// TIA Portal V20 export
VAR_GLOBAL   // PLC tag table "EasyBOX"
   I_OUT_TRAY1 AT %I31.0 : Bool;
   I_OUT_TRAY2 AT %I31.1 : Bool;
   I_OUT_TRAY3 AT %I31.2 : Bool;
   I_OUT_TRAY4 AT %I31.3 : Bool;
   I_OUT_TRAY5 AT %I31.4 : Bool;
   I_OUT_TRAY6 AT %I31.5 : Bool;
   I_OUT_TRAY7 AT %I31.6 : Bool;
   I_OUT_TRAY8 AT %I31.7 : Bool;
   I_OUT_TRAY9 AT %I33.0 : Bool;
   I_OUT_TRAY10 AT %I33.1 : Bool;
   I_OUT_TRAY11 AT %I33.2 : Bool;
   I_OUT_TRAY12 AT %I33.3 : Bool;
   ReqAccessAreaRobot AT %I33.4 : Bool;
   ResetAreaRobot AT %I33.5 : Bool;
   SB_Hold AT %I33.6 : Bool;   // Hold Button
   AIR_OK AT %I33.7 : Bool;
   SB_LockVice_MC1 AT %I35.0 : Bool;
   SB_LockPallet_MC1 AT %I35.1 : Bool;
   SB_LockVice_MC2 AT %I35.2 : Bool;
   SB_LockPallet_MC2 AT %I35.3 : Bool;
   SA_MC1_MANUAL AT %I35.4 : Bool;   // Selector keyboard on MC1 MANUAL
   SA_MC2_MANUAL AT %I35.5 : Bool;   // Selector keyboard on MC2 MANUAL
   All_trays_Inside AT %I35.6 : Bool;
   "free35.7" AT %I35.7 : Bool;
   HLStartAux AT %Q41.0 : Bool;
   HL_Hold AT %Q41.1 : Bool;
   HLReqAccess AT %Q41.2 : Bool;
   HLResetAccess AT %Q41.3 : Bool;
   HL_GREEN AT %Q41.4 : Bool;
   HL_ORANGE AT %Q41.5 : Bool;
   HL_RED AT %Q41.6 : Bool;
   HL_ViceClose_MC1 AT %Q41.7 : Bool;
   HL_palletLocked_MC1 AT %Q42.0 : Bool;
   HL_viceClose_MC2 AT %Q42.1 : Bool;
   HL_palletLocked_MC2 AT %Q42.2 : Bool;
   "free42.3" AT %Q42.3 : Bool;
   "free42.4" AT %Q42.4 : Bool;
   "free42.5" AT %Q42.5 : Bool;
   "free42.6" AT %Q42.6 : Bool;
   "free42.7" AT %Q42.7 : Bool;
   I_MC1_PalletLock AT %I43.7 : Bool;
   I_MC2_DoorOpen AT %I44.0 : Bool;
   I_MC2_ViceOpen AT %I44.1 : Bool;
   I_MC2_ViceClose AT %I44.2 : Bool;
   I_MC2_PalletUnlock AT %I44.3 : Bool;
   I_MC2_AutoMode AT %I44.4 : Bool;
   I_MC2_endWork AT %I44.5 : Bool;
   I_MC2_endClean AT %I44.6 : Bool;
   I_MC2_free AT %I44.7 : Bool;
   Q_MC1_LockPallet AT %Q45.5 : Bool;
   Q_MC1_OpenVice AT %Q45.2 : Bool;
   Q_MC1_CloseVice AT %Q45.3 : Bool;
   Q_MC1_UnlockPallet AT %Q45.4 : Bool;
   Q_MC1_StartWork AT %Q45.0 : Bool;
   Q_MC1_GateClosed AT %Q45.6 : Bool;
   Q_MC1_FuoriIngombro AT %Q45.1 : Bool;
   Q_MC1_free1 AT %Q45.7 : Bool;
   Q_MC2_OpenDoor AT %Q46.0 : Bool;
   Q_MC2_OpenVice AT %Q46.1 : Bool;
   Q_MC2_CloseVice AT %Q46.2 : Bool;
   Q_MC2_UnlockPallet AT %Q46.3 : Bool;
   Q_MC2_StartWork AT %Q46.4 : Bool;
   Q_MC2_StartClean AT %Q46.5 : Bool;
   Q_MC2_free AT %Q46.6 : Bool;
   Q_MC2_free1 AT %Q46.7 : Bool;
   I_MC1_DoorClosed AT %I43.2 : Bool;
   I_MC1_ViceOpened AT %I43.4 : Bool;
   I_MC1_ViceClosed AT %I43.5 : Bool;
   I_MC1_PalletUnlocked AT %I43.6 : Bool;
   I_MC1_AutoMode AT %I43.0 : Bool;
   I_MC1_EndWork AT %I43.1 : Bool;
   I_MC1_spare_3 AT %I43.3 : Bool;
END_VAR
